Staubli VAL3: Path11.pjx

--- Path11.pjx ---
Parameters version=s7.8.3 stackSize=5000 millimeterUnit=true
Program file=Delete.pgx
Program file=EditMain.pgx
Program file=EditPoint.pgx
Program file=EnterPageKey.pgx
Program file=getPtPara.pgx
Program file=Init.pgx
Program file=loadPath.pgx
Program file=Main.pgx
Program file=MainKey.pgx
Program file=OnF1.pgx
Program file=OnF2.pgx
Program file=OnF3.pgx
Program file=OnF4.pgx
Program file=OnF5.pgx
Program file=OnF6.pgx
Program file=OnF7.pgx
Program file=OnF8.pgx
Program file=readFileList.pgx
Program file=Refresh.pgx
Program file=Refresh1.pgx
Program file=Refresh2.pgx
Program file=Refresh3.pgx
Program file=RefreshList.pgx
Program file=Save.pgx
Program file=selectFile.pgx
Program file=SimuMain.pgx
Program file=start.pgx
Program file=stop.pgx
Data file=Path11.dtx
Library alias=master path=Disk://template/normal/normal.pjx
Library alias=user path=Disk://userPage/USERPAGE.pjx
Library alias=prd path=Disk://template/product/product.pjx
Library alias=PublicData path=Disk://PublicData/PublicData.pjx
Library alias=Tool path=Disk://Tool/Tool.pjx
Library alias=Frame path=Disk://Frame/Frame.pjx
Library alias=PublicProg path=Disk://PublicProg/PublicProg.pjx
Library alias=IO path=Disk://IO/IO.pjx
Library alias=SparePoint path=Disk://SparePoint/SparePoint.pjx

--- Main.pgx ---
program Main()
  local num l_nKey
begin
  //
  nPage=0
  do
    call Refresh()
    call RefreshList()
    call user:setList("路径",sList,bUserRefresh,bListRefresh,nSelected,sItem,l_nKey)
    bUserRefresh=false
    bListRefresh=false
    call MainKey(l_nKey)
    delay(0)
  until bExit

end

--- Delete.pgx ---
program Delete()
  local string l_sYesNo[2]
  local num l_i
begin
  //删除
  l_sYesNo[0]="是"
  l_sYesNo[1]="否"
  switch nPage
    case 0
      call user:questionDialog("是否删除此路径?",l_sYesNo,l_i)
      if l_i==0 or l_i==1
        if sFileList[nSelected]!=""
          libDelete(sFolder+sFileList[nSelected])
          delete(sFileList[nSelected])
          bListRefresh=true
        endIf
      endIf
    break
    case 1
      call user:questionDialog("是否删除此点?",l_sYesNo,l_i)
      if l_i==0 or l_i==1
        if sFileList[nSelected]!=""
          delete(prd:pDemo[nSelected])
          delete(prd:sPtParameter[nSelected])
          bListRefresh=true
        endIf
      endIf
    break
  endSwitch

  bUserRefresh=true
end

--- EditMain.pgx ---
public program EditMain(string x_sPath)
  local num l_nKey
  local bool l_bRes
begin
  //

  //
  //load path

    call loadPath(l_bRes,x_sPath)
    if !l_bRes
      return
    endIf

    //
    bUserRefresh=bListRefresh=true
    nPage=1
    //
    do
      call Refresh1()
      call RefreshList()
      call user:setList(x_sPath,sList,bUserRefresh,bListRefresh,nSelected,sItem,l_nKey)
      bUserRefresh=false
      bListRefresh=false
      call MainKey(l_nKey)
      delay(0)
    until bExit
    nPage=0
    bExit=false
    bUserRefresh=bListRefresh=true

end

--- EditPoint.pgx ---
program EditPoint()
  local bool l_bRes
  local num l_i
  local string l_sValue
  local num l_nSelect
  local string l_sItem
  local num l_nKey
  local num l_nRes
begin
  switch nPage
    //运动点
    case 1
      cls()
      resize(sParameter,1,11)
      sParameter[0]="X"
      sParameter[1]="Y"
      sParameter[2]="Z"
      sParameter[3]="Rx"
      sParameter[4]="Ry"
      sParameter[5]="Rz"
      sParameter[6]="P1"
      sParameter[7]="P2"
      sParameter[8]="IO1"
      sParameter[9]="IO2"
      sParameter[10]="delay"
      //
      resize(sListItemValue,1,size(sParameter))
      sListItemValue[0]=toString(".3",prd:pDemo[nSelected].trsf.x)
      sListItemValue[1]=toString(".3",prd:pDemo[nSelected].trsf.y)
      sListItemValue[2]=toString(".3",prd:pDemo[nSelected].trsf.z)
      sListItemValue[3]=toString(".3",prd:pDemo[nSelected].trsf.rx)
      sListItemValue[4]=toString(".3",prd:pDemo[nSelected].trsf.ry)
      sListItemValue[5]=toString(".3",prd:pDemo[nSelected].trsf.rz)
      //解析sPtParameter
      call getPtPara(prd:sPtParameter[nSelected],sPtPara)
      sListItemValue[6]=sPtPara[0]
      sListItemValue[7]=sPtPara[1]
      sListItemValue[8]=sPtPara[2]
      sListItemValue[9]=sPtPara[3]
      sListItemValue[10]=sPtPara[4]
      //
      for l_i=0 to size(sParameter)-1
        call user:strlength(sParameter[l_i],user:nBottomX/2)
        l_sValue=sListItemValue[l_i]
        call user:strlength(l_sValue,user:nBottomX/2+1)
        sParameter[l_i]=sParameter[l_i]+":"+l_sValue
      endFor

      bUserRefresh=true
      bListRefresh=true
      //
      do
        if bUserRefresh
          cls()
          call user:clear(0,13)
          call user:typeMenu(8,"确定")
        endIf
        call user:setList("编辑点",sParameter,bUserRefresh,bListRefresh,l_nSelect,l_sItem,l_nKey)
        bUserRefresh=false
        bListRefresh=false
        call EnterPageKey(l_nKey,l_nSelect,sParameter[l_nSelect])
        delay(0)
      until l_nKey==255 or l_nKey==278
      prd:sPtParameter[nSelected]=sListItemValue[6]+"/"+sListItemValue[7]+"/"+sListItemValue[8]+"/"+sListItemValue[9]+"/"+sListItemValue[10]
      bUserRefresh=true
      bListRefresh=true
    break
  endSwitch
end

--- EnterPageKey.pgx ---
program EnterPageKey(num& x_nKey, num& x_nSelect, string& x_sItem)
  local string l_sStr
  local num l_nKey
  local string l_sEmpty
  local string l_sValue
  local num l_nItem
  local num l_nView
  local string l_sItem
  local point lp
  local string l_sYN[2]
  local bool l_bRes
  local num l_nTemp
begin
  //
  //编辑项目
  switch x_nSelect
    //X
    case 0
      if x_nKey==270
        call user:editNum(x_sItem,sListItemValue[x_nSelect],prd:pDemo[nSelected].trsf.x,x_nSelect)
      endIf
    break
    //Y
    case 1
      if x_nKey==270
        call user:editNum(x_sItem,sListItemValue[x_nSelect],prd:pDemo[nSelected].trsf.y,x_nSelect)
      endIf
    break
    //Z
    case 2
      if x_nKey==270
        call user:editNum(x_sItem,sListItemValue[x_nSelect],prd:pDemo[nSelected].trsf.z,x_nSelect)
      endIf
    break
    //rx
    case 3
      if x_nKey==270
        call user:editNum(x_sItem,sListItemValue[x_nSelect],prd:pDemo[nSelected].trsf.rx,x_nSelect)
      endIf
    break
    //ry
    case 4
      if x_nKey==270
        call user:editNum(x_sItem,sListItemValue[x_nSelect],prd:pDemo[nSelected].trsf.ry,x_nSelect)
      endIf
    break
    //rz
    case 5
      if x_nKey==270
        call user:editNum(x_sItem,sListItemValue[x_nSelect],prd:pDemo[nSelected].trsf.rz,x_nSelect)
      endIf
    break
    //P1
    case 6
      if x_nKey==270
        call SparePoint:start()
        call SparePoint:getPoint(sListItemValue[x_nSelect])
        x_sItem="P1       :"+sListItemValue[x_nSelect]
      endIf

    break
    //P2
    case 7
      if x_nKey==270
        call SparePoint:start()
        call SparePoint:getPoint(sListItemValue[x_nSelect])
        x_sItem="P1       :"+sListItemValue[x_nSelect]
      endIf
    break
    //IO1
    case 8
      if x_nKey==270
        call IO:setIO(sListItemValue[x_nSelect])
        call IO:Main(1)
        call IO:getIO(sListItemValue[x_nSelect])
        //
        x_sItem="IO1      :"+sListItemValue[x_nSelect]
      endIf

    break
    //IO2
    case 9
      if x_nKey==270
        call IO:setIO(sListItemValue[x_nSelect])
        call IO:Main(1)
        call IO:getIO(sListItemValue[x_nSelect])
        //
        x_sItem="IO2      :"+sListItemValue[x_nSelect]
      endIf
    break
    //delay
    case 10
      if x_nKey==270
        call user:editNum(x_sItem,sListItemValue[x_nSelect],l_nTemp,x_nSelect)
      endIf
    break
  endSwitch
  if x_nKey==270
    bUserRefresh=true
    bListRefresh=true
  endIf
end

--- Init.pgx ---
program Init()
  local num l_ni
begin
  //
  bUserRefresh=bListRefresh=true
  //
  bExit=false
  //
  call readFileList(sFolder,sFileList)
  call selectFile(sDeli,sFileList)
  //

end

--- loadPath.pgx ---
program loadPath(bool& x_bRes, string x_sFile)
begin
  //加载路径
  x_bRes=false
  if prd:libLoad(sFolder+x_sFile)!=0
    logMsg(sItem+":加载失败")
    popUpMsg(sItem+":加载失败")
    return
  endIf
  x_bRes=true

end

--- MainKey.pgx ---
program MainKey(num x_nKey)
  local num l_nKey
begin
  //
  switch x_nKey
    //编辑
    case 271
      call OnF1()
    break
    //取反
    case 272
      call OnF2()
    break
    //删除
    case 273
      call OnF3()
    break
    //编辑
    case 274
      call OnF4()
    break
    //
    case 275
    break
    //
    case 276
      call OnF6()
    break
    //save
    case 277
      call OnF7()
    break
    //返回
    case 278
      call OnF8("是否返回")
    break
    case 270
      call EditPoint()
    break
  endSwitch
end

--- OnF1.pgx ---
program OnF1()
  local bool l_bRes
begin

  switch nPage
    case 0
      //编辑路径
      call EditMain(sItem)
    break
    case 1
      //
      tTool.trsf=Tool:tTool[prd:sToolName].trsf
      fFrame.trsf=Frame:fFrame[prd:sFrameName].trsf
      pTemp=here(tTool,fFrame)
      prd:pDemo[nSelected].trsf=pTemp.trsf
    break
    case 2

    break
    case 3
    break
    case 4
    break

  endSwitch
end

--- OnF2.pgx ---
program OnF2()
  local num l_ni
  local bool l_bRes
begin
  switch nPage
    case 0
      //模拟
      call SimuMain()
    break
    case 1
      //insert
      nSelected=nSelected+1
      insert(prd:pDemo[nSelected])
      prd:pDemo[nSelected]=here(Tool:tTool[prd:sToolName],Frame:fFrame[prd:sFrameName])
      insert(prd:sPtParameter[nSelected])
      //添加点的信息
    break
    case 2
    break
    case 3
    break
    case 4
    break

  endSwitch

end

--- OnF3.pgx ---
program OnF3()
begin
  //删除
  call Delete()
end

--- OnF4.pgx ---
program OnF4()
  local string l_sProperty[2]
  local string l_sItem
begin
  //调用tool or frame library
  l_sProperty[0]="工具"
  l_sProperty[1]="坐标系"
  call user:SetProerty("",26,9,6,2,l_sProperty,l_sItem)
  if l_sItem=="工具"
    call Tool:setTool(prd:sToolName)
    call Tool:Main(1)
    call Tool:getTool(prd:sToolName)
  elseIf l_sItem=="坐标系"
    call Frame:SetFrame(prd:sFrameName)
    call Frame:Main(1)
    call Frame:getFrame(prd:sFrameName)
  endIf
  bUserRefresh=bListRefresh=true
end

--- Refresh1.pgx ---
program Refresh1()
begin
  //编辑界面
  if bUserRefresh
    cls()
    userPage()
    gotoxy(1,1)
    put("F1->记录")
    gotoxy(1,13)
    put("F1")
    gotoxy(1,2)
    put("F2->插入")
    gotoxy(6,13)
    put("F2")
    gotoxy(1,3)
    put("F3->删除")
    gotoxy(11,13)
    put("F3")
    gotoxy(1,4)
    put("F4->选择工具/坐标系")
    gotoxy(16,13)
    put("F4")

    gotoxy(1,5)
    put("F5->运动方向切换")
    gotoxy(21,13)
    put("F5")
    //    gotoxy(1,6)
    //    put("F6->")
    //    gotoxy(26,13)
    //    put("")
    gotoxy(1,7)
    put("F7->保存")
    gotoxy(31,13)
    put("F7")
    gotoxy(1,8)
    put("F8->返回")
    gotoxy(36,13)
    put("F8")

    //
    gotoxy(1,10)
    put("工具："+prd:sToolName)
    gotoxy(1,11)
    put("坐标系："+prd:sFrameName)
  endIf
end

--- selectFile.pgx ---
public program selectFile(string& x_sDelimiter[], string& x_sList[])
  local num l_ni
  local num l_nj
begin
  //
  for l_nj=0 to size(x_sList)-1
    if x_sList[l_ni]!=""
      for l_ni=0 to size(x_sDelimiter)-1
        if left(x_sList[l_nj],1)==x_sDelimiter[l_ni]
          l_ni=size(x_sDelimiter)
        endIf
        if l_ni==size(x_sDelimiter)-1
          delete(x_sList[l_nj])
          l_nj=l_nj-1
        endIf
      endFor
    endIf

  endFor
end

--- SimuMain.pgx ---
program SimuMain()
  local num l_nKey
begin
  //
  nPage=2
  bUserRefresh=bListRefresh=true
  do
    call Refresh2()
    call RefreshList()
    call user:setList("路径",sList,bUserRefresh,bListRefresh,nSelected,sItem,l_nKey)
    bUserRefresh=false
    bListRefresh=false
    call MainKey(l_nKey)
    delay(0)
  until bExit
  nPage=0
  bUserRefresh=bListRefresh=true
  bExit=false
end
